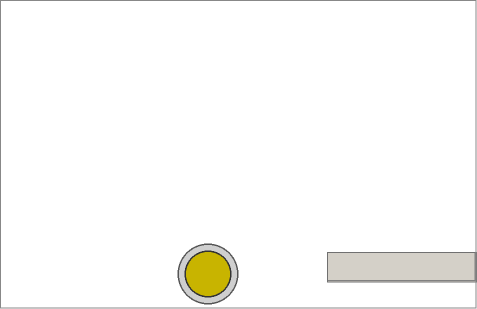
VISUALIZATION Visualization_1  // 477x309
    Button (327,252 150x30)
        OnMouseDown: toggle Variables.Button
        OnMouseUp: toggle Variables.Button
    Lamp1 (173,239 70x70), variable: Variables.LED, style: Lamp-Lamp1-Yellow
END_VISUALIZATION

(* stored: Version 1.1.0.1, ProductVersion 3.1.4024.12
   Visu Visualization_1: Id {d3168e93-4af8-4970-8467-d44ac00688da} *)
